PROGRAM MAIN
VAR
	//blockgolf1: FB_Blokgolf;
	_product1: ST_ProductInfo := (eproductType := E_ProductType.cube, fDimension1 := 10, fDimension2 := 5, fDimension3 := 12, fSpecificWeight := 1000);
	_product2: ST_ProductInfo := (eproductType := E_ProductType.cylinder, fDimension1 := 20, fDimension2 := 10, fDimension3 := 24, fSpecificWeight := 2000);
	inventory1: FB_Inventory(product1 := _product1, product2 := _product2);
	bTest: BOOL;

END_VAR

IF bTest THEN
	inventory1.M_Add(_product2);
	inventory1.M_Remove(0);
	bTest := FALSE;
END_IF

END_PROGRAM

(* stored: Version 1.1.0.1, ProductVersion 3.1.4024.13
   POU MAIN: Id {7de039f4-eca8-4806-a063-3ce089714fb6}, SpecialFunc None *)
